FUNCTION_BLOCK PalletizerConveyor EXTENDS Conveyor
VAR_INPUT
END_VAR
VAR_OUTPUT
	bStartBackward : BOOL;
END_VAR
VAR	
	fbStartBackward : BoolOut;
END_VAR

SUPER^();
bStartBackward := fbStartBackward.getValue;

PROPERTY getStartBackward : I_StepCondition
GET
getStartBackward := fbStartBackward;
END_GET
END_PROPERTY

END_FUNCTION_BLOCK

(* stored: Version 1.1.0.1, ProductVersion 3.1.4024.2
   POU PalletizerConveyor: Id {2ce7a42e-b441-4b88-9e0a-c833ce71c0d4}, SpecialFunc None
   Property getStartBackward: Id {1be61ee4-2b11-41d3-b441-0dd528ef6733}
   Get Get: Id {08cd3fdd-45df-4c96-8883-2d6eba7e8d6b} *)
